// TwinCAT 3 PLC project PLC_TMO_VAC_FS
// ProgramVersion: 3.1.4022.7
// libraries:
//   L2SI Vacuum Library, * (SLAC)
//   LCLS General, * (SLAC)
//   PMPS, * (SLAC - LCLS)
//   Tc2_Standard, * (Beckhoff Automation GmbH)
//   Tc2_System, * (Beckhoff Automation GmbH)
//   Tc3_Module, * (Beckhoff Automation GmbH)
// project tree:
//   GVLs/ GVL_FS.TcGVL
//   / PlcTask.TcTTO (not stored)
//   POUs/ MAIN.TcPOU
// (motion and I/O tree: see PLC project plc_tmo_vac)
// real-time tasks:
//   TASK PlcTask: cycle T#10ms, priority 20, ADS port 350
// variable links:

// ---- GVLs/GVL_FS.TcGVL
//{attribute 'qualified_only'}
VAR_GLOBAL
	
	{attribute 'TcLinkTo' := 	'.i_xOPNLS	:=	TIIB[K4S20-E1-FSV (EL1004)]^Channel 2^Input;
								 .i_xClsLS	:=	TIIB[K4S20-E1-FSV (EL1004)]^Channel 1^Input;
								 .q_xClose_A	:=	TIIB[K4S20-E2-FSV (EL2202)]^Channel 1^Output;
								 .q_xClose_B	:=	TIIB[K4S20-E2-FSV (EL2202)]^Channel 2^Output;
								 .q_xClose_C	:=	TIIB[K4S20-E3-FSV (EL2202)]^Channel 1^Output;
								 .q_xOPN_DO		:=	TIIB[K4S20-E3-FSV (EL2202)]^Channel 2^Output;
								 .i_xTrigger	:= TIIB[R20_EK0_E5 (EL1124)]^Channel 1^Input
								 
	'}
	{attribute 'pytmc' := '
		pv: TV1K4:VFS:01
		
	'}
	TV1K4_VFS_01 : FB_VFS;
	GCC : FB_MKS500_EP;
	

END_VAR

// ---- POUs/MAIN.TcPOU
PROGRAM MAIN
VAR
	i_xFFReset: INT;
END_VAR

TV1K4_VFS_01(
	i_xPMPS_OK:= TRUE, 
	i_xExt_OK:= TRUE, 
	i_xOverrideMode:= FALSE, 
	iq_stValve=> );

END_PROGRAM
